Staubli VAL3: destroyAdvMoves.pgx

program destroyAdvMoves()
  local num l_nIndex
begin

  //setMutex(bAdvMoves)
  for l_nIndex=0 to size(bAdvMoveBusy)-1
    if bAdvMoveBusy[l_nIndex]
      taskKill(sAdvMovePrefix+toString("",l_nIndex))
      wait(taskStatus(sAdvMovePrefix+toString("",l_nIndex))==-1)
      bAdvMoveBusy[l_nIndex]=false
    endIf
  endFor
  //bAdvMoves=false

end
